(*udt (user defined type) of Beckhoff Type EtherCAT Master:
	auth. Brent Lekx-Toniolo of Toniolo Research & Development Inc.; 
	July 2010; version 1.0*)



TYPE udt_ECATMaster_Status :
STRUCT
	Frm0State: UINT;
	(*
	0x0001 = 1. EtherCAT command NOT sent (NOP requested)
	0x0002 = 2. EtherCAT command NOT sent (NOP requested)
	0x0004 = 3. EtherCAT command NOT sent (NOP requested)
	...
	0x4000 = 15. EtherCAT command NOT sent (NOP requested)
	0x8000 = complete frame NOT sent*)
	Frm0WcState: UINT;
	(*
	0x0001 = wrong working counter of 1. EtherCAT command received
	0x0002 = wrong working counter of 2. EtherCAT command received
	0x0004 = wrong working counter of 3. EtherCAT command received
	...
	0x4000 = wrong working counter of 15. EtherCAT command received
	0x8000 = complete frame missing*)
	FR5State: UINT;
	(*
	0x0001 = 1. EtherCAT command NOT sent (NOP requested)
	0x0002 = 2. EtherCAT command NOT sent (NOP requested)
	0x0004 = 3. EtherCAT command NOT sent (NOP requested)
	...
	0x4000 = 15. EtherCAT command NOT sent (NOP requested)
	0x8000 = complete frame NOT sent*)
	FR5WcState: UINT;
	(*
	0x0001 = wrong working counter of 1. EtherCAT command received
	0x0002 = wrong working counter of 2. EtherCAT command received
	0x0004 = wrong working counter of 3. EtherCAT command received
	...
	0x4000 = wrong working counter of 15. EtherCAT command received
	0x8000 = complete frame missing*)
	FR7State: UINT;
	(*
	0x0001 = 1. EtherCAT command NOT sent (NOP requested)
	0x0002 = 2. EtherCAT command NOT sent (NOP requested)
	0x0004 = 3. EtherCAT command NOT sent (NOP requested)
	...
	0x4000 = 15. EtherCAT command NOT sent (NOP requested)
	0x8000 = complete frame NOT sent*)
	FR7WcState: UINT;
	(*
	0x0001 = wrong working counter of 1. EtherCAT command received
	0x0002 = wrong working counter of 2. EtherCAT command received
	0x0004 = wrong working counter of 3. EtherCAT command received
	...
	0x4000 = wrong working counter of 15. EtherCAT command received
	0x8000 = complete frame missing*)
	FR9State: UINT;
	(*
	0x0001 = 1. EtherCAT command NOT sent (NOP requested)
	0x0002 = 2. EtherCAT command NOT sent (NOP requested)
	0x0004 = 3. EtherCAT command NOT sent (NOP requested)
	...
	0x4000 = 15. EtherCAT command NOT sent (NOP requested)
	0x8000 = complete frame NOT sent*)
	FR9WcState: UINT;
	(*
	0x0001 = wrong working counter of 1. EtherCAT command received
	0x0002 = wrong working counter of 2. EtherCAT command received
	0x0004 = wrong working counter of 3. EtherCAT command received
	...
	0x4000 = wrong working counter of 15. EtherCAT command received
	0x8000 = complete frame missing*)

	SlaveCount: UINT;
	(*
	Actual count of EtherCAT slaves received*)

	DevState: UINT;
	(*
	0x0001 = Link error
	0x0002 = I/O locked after link error (I/O reset required)
	0x0004 = Link error (redundancy adapter)
	0x0008 = Missing one frame (redundancy mode)
	0x0010 = Out of send resources (I/O reset required)
	0x0020 = Watchdog triggered
	0x0040 = Ethernet driver (miniport) not found
	0x0080 = I/O reset active
	0x0100 = At least one device in 'INIT' state
	0x0200 = At least one device in 'PRE-OP' state
	0x0400 = At least one device in 'SAFE-OP' state
	0x0800 = At least one device indicates an error state
	0x1000 = DC not in sync*)

	CfgSlaveCount: UINT;
	(*
	Count of configured EtherCAT slaves
	*)
END_STRUCT
END_TYPE

(* stored: Version 1.1.0.1, ProductVersion 3.1.4024.9
   DUT udt_ECATMaster_Status: Id {5a441158-61b9-4499-8aa0-a2ef04b7f080} *)
